// TIA Portal V18 program export: 8 tag tables, 0 data types, 0 data blocks, 7 code blocks (in call order from the OBs), 0 instance data blocks

VAR_GLOBAL   // PLC tag table "Default tag table"
   System_Byte AT %MB1 : Byte;
   FirstScan AT %M1.0 : Bool;
   DiagStatusUpdate AT %M1.1 : Bool;
   AlwaysTRUE AT %M1.2 : Bool;
   AlwaysFALSE AT %M1.3 : Bool;
   Clock_Byte AT %MB0 : Byte;
   Clock_10Hz AT %M0.0 : Bool;
   Clock_5Hz AT %M0.1 : Bool;
   "Clock_2.5Hz" AT %M0.2 : Bool;
   Clock_2Hz AT %M0.3 : Bool;
   "Clock_1.25Hz" AT %M0.4 : Bool;
   Clock_1Hz AT %M0.5 : Bool;
   "Clock_0.625Hz" AT %M0.6 : Bool;
   "Clock_0.5Hz" AT %M0.7 : Bool;
   PTRIG AT %M2.0 : Bool;
   PTRIG2 AT %M2.1 : Bool;
END_VAR

VAR_GLOBAL   // PLC tag table "INPUT"
   I_Mode AT %I0.0 : Bool;   // Switch chế độ 1 auto, 0 manu
   I_CB_Cao AT %I0.1 : Bool;   // Cảm biến sản phẩm cao
   I_CB_Trung_Binh AT %I0.2 : Bool;   // Cảm biến sản phẩm trung bình
   I_CB_Thap AT %I0.3 : Bool;   // Cảm biến sản phẩm thấp
   I_BT AT %I0.4 : Bool;   // Chạy/Dừng động cơ băng tải
   I_Xylanh_Cao AT %I0.5 : Bool;   // Đóng/mở xi lanh sản phẩm cao
   I_Xylanh_TB AT %I0.6 : Bool;   // Đóng/mở xi lanh sản phẩm trung bình
END_VAR

VAR_GLOBAL   // PLC tag table "INPUT_M"
   M_Mode AT %M10.0 : Bool;   // Switch chế độ 1 auto, 0 manu
   M_CB_Cao AT %M10.1 : Bool;   // Cảm biến sản phẩm cao
   M_CB_Trung_Binh AT %M10.2 : Bool;   // Cảm biến sản phẩm trung bình
   M_CB_Thap AT %M10.3 : Bool;   // Cảm biến sản phẩm thấp
   M_BT AT %M10.4 : Bool;   // Chạy/Dừng động cơ băng tải
   M_Xylanh_Cao AT %M10.5 : Bool;   // Đóng/mở xi lanh sản phẩm cao
   M_Xylanh_TB AT %M10.6 : Bool;   // Đóng/mở xi lanh sản phẩm trung bình
END_VAR

VAR_GLOBAL   // PLC tag table "OUTPUT"
   Q_lamp_Auto AT %Q0.0 : Bool;   // Đèn chế độ auto
   Q_lamp_Manu AT %Q0.1 : Bool;   // Đèn chế độ manu
   Q_BT AT %Q0.2 : Bool;   // Băng tải phân loại
   Q_Xylanh_Cao AT %Q0.3 : Bool;   // Xi lanh đẩy sản phẩm cao
   Q_Xylanh_TB AT %Q0.4 : Bool;   // Xi lanh đẩy sản phẩm trung bình
END_VAR

VAR_GLOBAL   // PLC tag table "PTRIG"
   P1 AT %M330.0 : Bool;
   P2 AT %M330.1 : Bool;
   P3 AT %M330.2 : Bool;
   P4 AT %M330.3 : Bool;
   P5 AT %M330.4 : Bool;
   P6 AT %M330.5 : Bool;
   P7 AT %M330.6 : Bool;
   P8 AT %M330.7 : Bool;
   P9 AT %M331.0 : Bool;
   P10 AT %M331.1 : Bool;
   P11 AT %M331.2 : Bool;
END_VAR

VAR_GLOBAL   // PLC tag table "SO_NGUYEN"
   Act_Count_Cao AT %MW200 : Int;   // Bộ đếm số sản phẩm trọng lượng nhẹ
   Act_Count_TB AT %MW202 : Int;   // Bộ đếm số sản phẩm trọng lượng trung bình
   Act_Count_Thap AT %MW204 : Int;   // Bộ đếm số sản phẩm trọng lượng nặng
   Simu_VT_SP AT %MW206 : Int;   // Mô phỏng vị trí sản phẩm
   Simu_Type_SP AT %MW208 : Int;   // Mô phỏng loại sản phẩm
END_VAR

VAR_GLOBAL   // PLC tag table "TAG"
   Start AT %I0.0 : Bool;   // Nút nhấn Start
   Stop AT %I0.1 : Bool;   // Nút nhấn Stop
   Lamp AT %Q0.0 : Bool;   // Đèn hệ thống làm việc
   Sensor_Temperature AT %IW64 : Int;   // Cảm biến nhiệt độ
   QW_SSR AT %QW64 : Int;   // Đầu ra analog điều khiển SSR
   HMI_Start AT %M10.0 : Bool;   // Nút nhấn start trên Scada
   HMI_Stop AT %M10.1 : Bool;   // Nút nhấn Stop trên Scada
   HMI_Simulation AT %M10.2 : Bool;   // Nút mô phỏng tín hiệu nhiệt độ trên Scada
   HMI_Simu_Temperature AT %MW100 : Int;   // Mô phỏng nhiệt độ trên HMI
   HMI_Setting_Temperature AT %MD200 : Real;   // Cài đặt nhiệt độ cho máy sấy
   HMI_TT_Temperature AT %MD204 : Real;   // Nhiệt độ thực tế máy sấy
END_VAR

VAR_GLOBAL   // PLC tag table "TRUNGGIAN"
   Q_Auto_BT AT %M20.0 : Bool;   // Băng tải phân loại
   Q_Auto_Xylanh_Cao AT %M20.1 : Bool;   // Xi lanh đẩy sản phẩm cao
   Q_Auto_Xylanh_TB AT %M20.2 : Bool;   // Xi lanh đẩy sản phẩm trung bình
   Q_Manu_BT AT %M30.0 : Bool;   // Băng tải phân loại
   Q_Manu_Xylanh_Cao AT %M30.1 : Bool;   // Xi lanh đẩy sản phẩm cao
   Q_Manu_Xylanh_TB AT %M30.2 : Bool;   // Xi lanh đẩy sản phẩm trung bình
   M_Simulation AT %M5.0 : Bool;   // Nút mô phỏng trên scada
   M_Reset AT %M5.1 : Bool;   // Nút reset
   SIMU_CB_CAO AT %M5.2 : Bool;   // Mô phỏng cảm biến cao
   SIMU_CB_TB AT %M5.3 : Bool;   // Mô phỏng cảm biến trung bình
   SIMU_CB_THAP AT %M5.4 : Bool;   // Mô phỏng cảm biến thấp
END_VAR

ORGANIZATION_BLOCK "Main"   // OB1, LAD, ProgramCycle
TITLE = "Main Program Sweep (Cycle)"
{ S7_Optimized_Access := 'TRUE' }
VERSION : 0.1
// stored: AutoNumber true, IsIECCheckEnabled false, SetENOAutomatically false
   VAR_INPUT
      Initial_Call : Bool;   // Initial call of this OB
      Remanence : Bool;   // =True, if remanent data are available
   END_VAR
   VAR_TEMP
      TG_ND : Int;
      TG_ND1 : Real;
   END_VAR
BEGIN

REGION Network 1: Điều khiển đèn làm việc
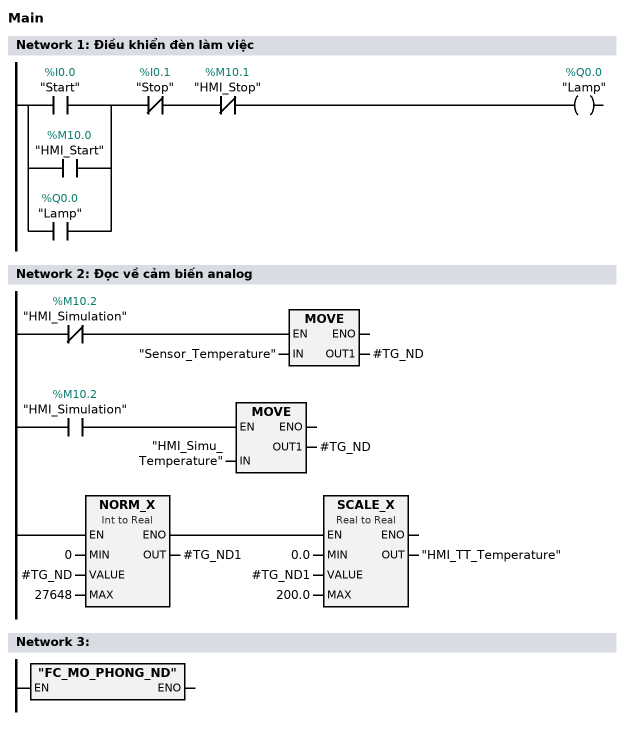
   RUNG wire#powerrail
      Contact( "Start" )
      wire#w1
      I_Contact( "Stop" )
      I_Contact( "HMI_Stop" )
      Coil( "Lamp" )
   END_RUNG
   RUNG wire#powerrail
      Contact( "HMI_Start" )
   END_RUNG wire#w1
   RUNG wire#powerrail
      Contact( "Lamp" )
   END_RUNG wire#w1
   // the same network as SCL:
   "Lamp" := ("Start" OR "HMI_Start" OR "Lamp") AND NOT "Stop" AND NOT "HMI_Stop";
END_REGION

REGION Network 2: Đọc về cảm biến analog
   RUNG wire#powerrail
      I_Contact( "HMI_Simulation" )
      Move(in := "Sensor_Temperature", out1 => #TG_ND)
   END_RUNG
   RUNG wire#powerrail
      Contact( "HMI_Simulation" )
      Move(in := "HMI_Simu_Temperature", out1 => #TG_ND)
   END_RUNG
   RUNG wire#powerrail
      { S7_Templates := "[SrcType := Int, DestType := Real]" } Normalize(min := 0, value := #TG_ND, max := 27648, out => #TG_ND1)
      { S7_Templates := "[SrcType := Real, DestType := Real]" } Scale(min := 0.0, value := #TG_ND1, max := 200.0, out => "HMI_TT_Temperature")
   END_RUNG
   // the same network as SCL:
   IF NOT "HMI_Simulation" THEN #TG_ND := "Sensor_Temperature"; END_IF;
   IF "HMI_Simulation" THEN #TG_ND := "HMI_Simu_Temperature"; END_IF;
   #TG_ND1 := NORM_X(MIN := 0, VALUE := #TG_ND, MAX := 27648);
   "HMI_TT_Temperature" := SCALE_X(MIN := 0.0, VALUE := #TG_ND1, MAX := 200.0);
END_REGION

REGION Network 3
   RUNG wire#powerrail
      "FC_MO_PHONG_ND"()
   END_RUNG
   // the same network as SCL:
   "FC_MO_PHONG_ND"();
END_REGION
END_ORGANIZATION_BLOCK

FUNCTION "FC_MO_PHONG_ND" : Void   // FC1, LAD
{ S7_Optimized_Access := 'TRUE' }
VERSION : 0.1
// stored: AutoNumber true, IsIECCheckEnabled false, SetENOAutomatically false, UDAEnableTagReadback false
   VAR_TEMP   // added for the SCL form of the ladder/FBD networks
      _w1 : Bool;
      _w2 : Bool;
      _w3 : Bool;
      _w4 : Bool;
   END_VAR
BEGIN

REGION Network 1
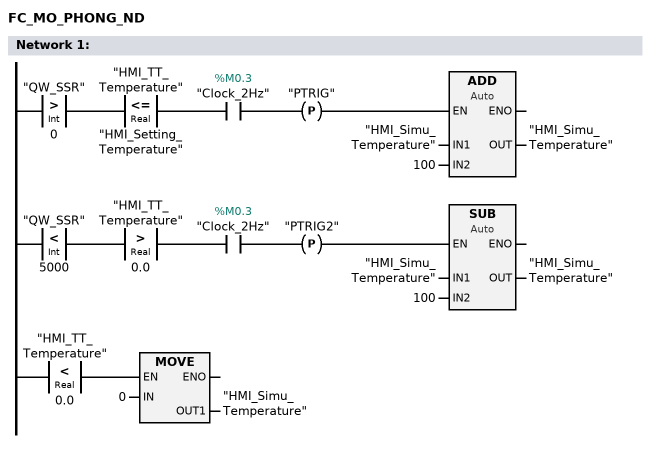
   RUNG wire#powerrail
      { S7_Templates := "SrcType := Int" } GT_Contact(in1 := "QW_SSR", in2 := 0)
      { S7_Templates := "SrcType := Real" } LE_Contact(in1 := "HMI_TT_Temperature", in2 := "HMI_Setting_Temperature")
      Contact( "Clock_2Hz" )
      P_Trig( "PTRIG" )
      Add(in1 := "HMI_Simu_Temperature", in2 := 100, out => "HMI_Simu_Temperature")
   END_RUNG
   RUNG wire#powerrail
      { S7_Templates := "SrcType := Int" } LT_Contact(in1 := "QW_SSR", in2 := 5000)
      { S7_Templates := "SrcType := Real" } GT_Contact(in1 := "HMI_TT_Temperature", in2 := 0.0)
      Contact( "Clock_2Hz" )
      P_Trig( "PTRIG2" )
      Sub(in1 := "HMI_Simu_Temperature", in2 := 100, out => "HMI_Simu_Temperature")
   END_RUNG
   RUNG wire#powerrail
      { S7_Templates := "SrcType := Real" } LT_Contact(in1 := "HMI_TT_Temperature", in2 := 0.0)
      Move(in := 0, out1 => "HMI_Simu_Temperature")
   END_RUNG
   // the same network as SCL:
   #_w1 := ("QW_SSR" > 0) AND ("HMI_TT_Temperature" <= "HMI_Setting_Temperature") AND "Clock_2Hz";
   #_w2 := #_w1 AND NOT "PTRIG";   // rising edge
   "PTRIG" := #_w1;
   IF #_w2 THEN "HMI_Simu_Temperature" := "HMI_Simu_Temperature" + 100; END_IF;
   #_w3 := ("QW_SSR" < 5000) AND ("HMI_TT_Temperature" > 0.0) AND "Clock_2Hz";
   #_w4 := #_w3 AND NOT "PTRIG2";   // rising edge
   "PTRIG2" := #_w3;
   IF #_w4 THEN "HMI_Simu_Temperature" := "HMI_Simu_Temperature" - 100; END_IF;
   IF "HMI_TT_Temperature" < 0.0 THEN "HMI_Simu_Temperature" := 0; END_IF;
END_REGION
END_FUNCTION

ORGANIZATION_BLOCK "Cyclic interrupt"   // OB30, LAD, CyclicInterrupt
{ S7_Optimized_Access := 'TRUE' }
VERSION : 0.1
// stored: AutoNumber true, IsIECCheckEnabled false, SetENOAutomatically false
   VAR_INPUT
      Initial_Call : Bool;   // Initial call of this OB
      Event_Count : Int;   // Events discarded
   END_VAR
BEGIN

REGION Network 1
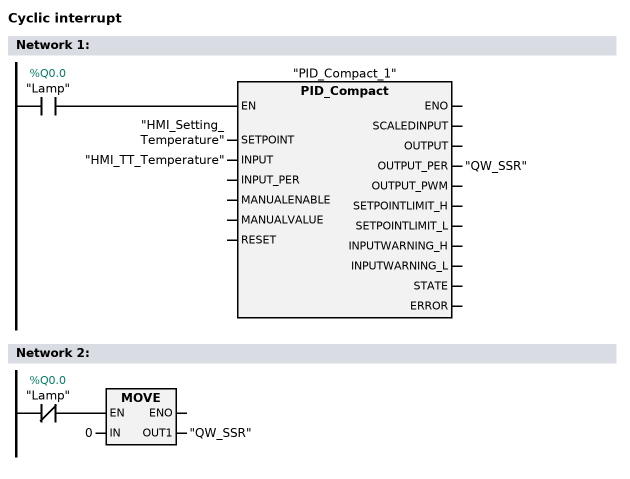
   RUNG wire#powerrail
      Contact( "Lamp" )
      "PID_Compact_1".PID_Compact(Setpoint := "HMI_Setting_Temperature", Input := "HMI_TT_Temperature", Input_PER :=, ManualEnable :=, ManualValue :=, Reset :=, ScaledInput =>, Output =>, Output_PER => "QW_SSR", Output_PWM =>, SetpointLimit_H =>, SetpointLimit_L =>, InputWarning_H =>, InputWarning_L =>, State =>, Error =>)
   END_RUNG
   // the same network as SCL:
   IF "Lamp" THEN
       "PID_Compact_1"(Setpoint := "HMI_Setting_Temperature", Input := "HMI_TT_Temperature", Output_PER => "QW_SSR");   // PID_Compact
   END_IF;
END_REGION

REGION Network 2
   RUNG wire#powerrail
      I_Contact( "Lamp" )
      Move(in := 0, out1 => "QW_SSR")
   END_RUNG
   // the same network as SCL:
   IF NOT "Lamp" THEN "QW_SSR" := 0; END_IF;
END_REGION
END_ORGANIZATION_BLOCK

FUNCTION "FC_AUTO_MODE" : Void   // FC2, LAD
{ S7_Optimized_Access := 'TRUE' }
VERSION : 0.1
// stored: AutoNumber true, IsIECCheckEnabled false, SetENOAutomatically false, UDAEnableTagReadback false
   VAR_TEMP   // added for the SCL form of the ladder/FBD networks
      _w1 : Bool;
      _w2 : Bool;
      _w3 : Bool;
      _w4 : Bool;
      _w5 : Bool;
      _w6 : Bool;
   END_VAR
BEGIN

REGION Network 1: RESET CÁC BỘ ĐẾM VỀ 0
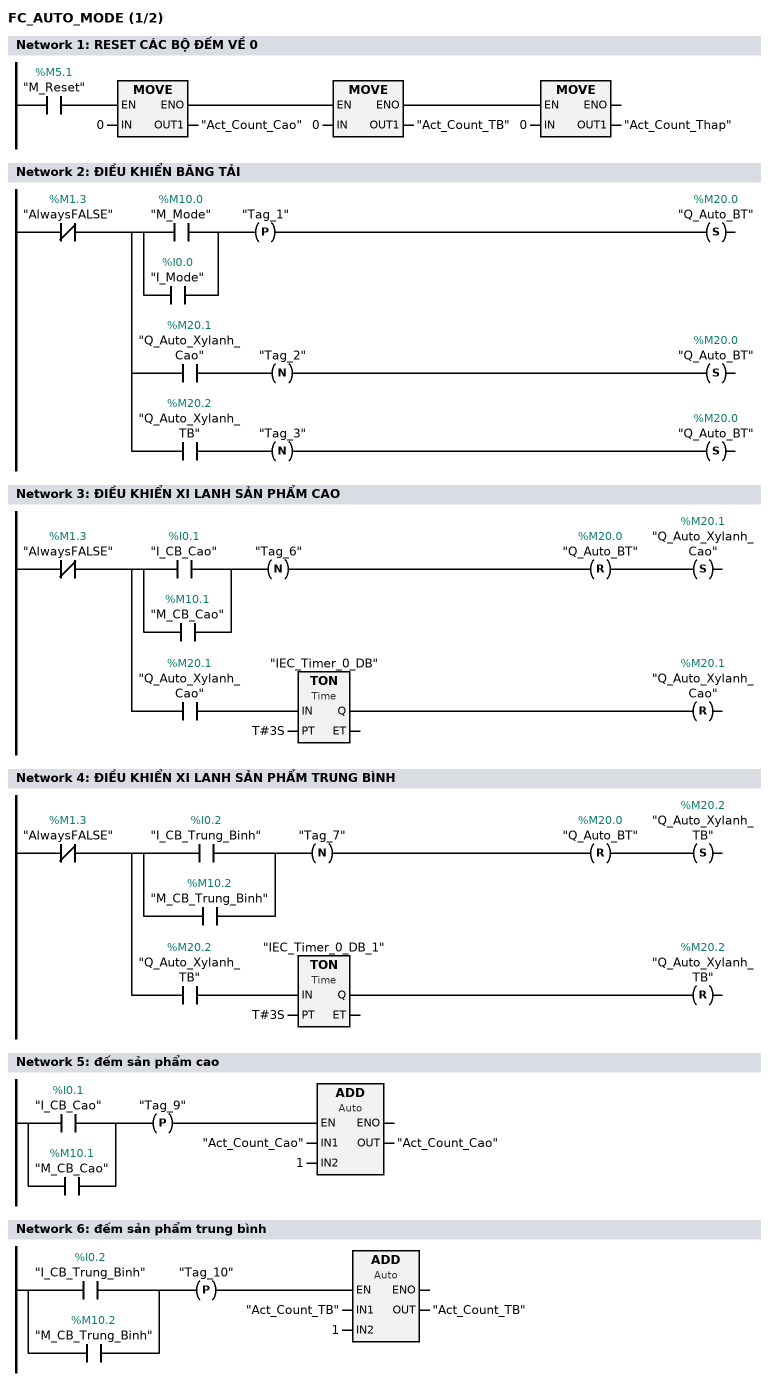
   RUNG wire#powerrail
      Contact( "M_Reset" )
      Move(in := 0, out1 => "Act_Count_Cao")
      Move(in := 0, out1 => "Act_Count_TB")
      Move(in := 0, out1 => "Act_Count_Thap")
   END_RUNG
   // the same network as SCL:
   IF "M_Reset" THEN
       "Act_Count_Cao" := 0;
       "Act_Count_TB" := 0;
       "Act_Count_Thap" := 0;
   END_IF;
END_REGION

REGION Network 2: ĐIỀU KHIỂN BĂNG TẢI
   RUNG wire#powerrail
      I_Contact( "AlwaysFALSE" )
      wire#w1
      Contact( "M_Mode" )
      wire#w2
      P_Trig( "Tag_1" )
      S_Coil( "Q_Auto_BT" )
   END_RUNG
   RUNG wire#w1
      Contact( "I_Mode" )
   END_RUNG wire#w2
   RUNG wire#w1
      Contact( "Q_Auto_Xylanh_Cao" )
      N_Trig( "Tag_2" )
      S_Coil( "Q_Auto_BT" )
   END_RUNG
   RUNG wire#w1
      Contact( "Q_Auto_Xylanh_TB" )
      N_Trig( "Tag_3" )
      S_Coil( "Q_Auto_BT" )
   END_RUNG
   // the same network as SCL:
   #_w1 := NOT "AlwaysFALSE" AND ("M_Mode" OR "I_Mode");
   #_w2 := #_w1 AND NOT "Tag_1";   // rising edge
   "Tag_1" := #_w1;
   IF #_w2 THEN "Q_Auto_BT" := TRUE; END_IF;
   #_w3 := NOT "AlwaysFALSE" AND "Q_Auto_Xylanh_Cao";
   #_w4 := NOT #_w3 AND "Tag_2";   // falling edge
   "Tag_2" := #_w3;
   IF #_w4 THEN "Q_Auto_BT" := TRUE; END_IF;
   #_w5 := NOT "AlwaysFALSE" AND "Q_Auto_Xylanh_TB";
   #_w6 := NOT #_w5 AND "Tag_3";   // falling edge
   "Tag_3" := #_w5;
   IF #_w6 THEN "Q_Auto_BT" := TRUE; END_IF;
END_REGION

REGION Network 3: ĐIỀU KHIỂN XI LANH SẢN PHẨM CAO
   RUNG wire#powerrail
      I_Contact( "AlwaysFALSE" )
      wire#w1
      Contact( "I_CB_Cao" )
      wire#w2
      N_Trig( "Tag_6" )
      R_Coil( "Q_Auto_BT" )
      S_Coil( "Q_Auto_Xylanh_Cao" )
   END_RUNG
   RUNG wire#w1
      Contact( "M_CB_Cao" )
   END_RUNG wire#w2
   RUNG wire#w1
      Contact( "Q_Auto_Xylanh_Cao" )
      { S7_Templates := "time_type := Time" } "IEC_Timer_0_DB".TON(pt := T#3S, et =>)
      R_Coil( "Q_Auto_Xylanh_Cao" )
   END_RUNG
   // the same network as SCL:
   #_w1 := NOT "AlwaysFALSE" AND ("I_CB_Cao" OR "M_CB_Cao");
   #_w2 := NOT #_w1 AND "Tag_6";   // falling edge
   "Tag_6" := #_w1;
   IF #_w2 THEN
       "Q_Auto_BT" := FALSE;
       "Q_Auto_Xylanh_Cao" := TRUE;
   END_IF;
   "IEC_Timer_0_DB".TON(IN := NOT "AlwaysFALSE" AND "Q_Auto_Xylanh_Cao", PT := T#3S);
   IF "IEC_Timer_0_DB".Q THEN "Q_Auto_Xylanh_Cao" := FALSE; END_IF;
END_REGION

REGION Network 4: ĐIỀU KHIỂN XI LANH SẢN PHẨM TRUNG BÌNH
   RUNG wire#powerrail
      I_Contact( "AlwaysFALSE" )
      wire#w1
      Contact( "I_CB_Trung_Binh" )
      wire#w2
      N_Trig( "Tag_7" )
      R_Coil( "Q_Auto_BT" )
      S_Coil( "Q_Auto_Xylanh_TB" )
   END_RUNG
   RUNG wire#w1
      Contact( "M_CB_Trung_Binh" )
   END_RUNG wire#w2
   RUNG wire#w1
      Contact( "Q_Auto_Xylanh_TB" )
      { S7_Templates := "time_type := Time" } "IEC_Timer_0_DB_1".TON(pt := T#3S, et =>)
      R_Coil( "Q_Auto_Xylanh_TB" )
   END_RUNG
   // the same network as SCL:
   #_w1 := NOT "AlwaysFALSE" AND ("I_CB_Trung_Binh" OR "M_CB_Trung_Binh");
   #_w2 := NOT #_w1 AND "Tag_7";   // falling edge
   "Tag_7" := #_w1;
   IF #_w2 THEN
       "Q_Auto_BT" := FALSE;
       "Q_Auto_Xylanh_TB" := TRUE;
   END_IF;
   "IEC_Timer_0_DB_1".TON(IN := NOT "AlwaysFALSE" AND "Q_Auto_Xylanh_TB", PT := T#3S);
   IF "IEC_Timer_0_DB_1".Q THEN "Q_Auto_Xylanh_TB" := FALSE; END_IF;
END_REGION

REGION Network 5: đếm sản phẩm cao
   RUNG wire#powerrail
      Contact( "I_CB_Cao" )
      wire#w1
      P_Trig( "Tag_9" )
      Add(in1 := "Act_Count_Cao", in2 := 1, out => "Act_Count_Cao")
   END_RUNG
   RUNG wire#powerrail
      Contact( "M_CB_Cao" )
   END_RUNG wire#w1
   // the same network as SCL:
   #_w1 := "I_CB_Cao" OR "M_CB_Cao";
   #_w2 := #_w1 AND NOT "Tag_9";   // rising edge
   "Tag_9" := #_w1;
   IF #_w2 THEN "Act_Count_Cao" := "Act_Count_Cao" + 1; END_IF;
END_REGION

REGION Network 6: đếm sản phẩm trung bình
   RUNG wire#powerrail
      Contact( "I_CB_Trung_Binh" )
      wire#w1
      P_Trig( "Tag_10" )
      Add(in1 := "Act_Count_TB", in2 := 1, out => "Act_Count_TB")
   END_RUNG
   RUNG wire#powerrail
      Contact( "M_CB_Trung_Binh" )
   END_RUNG wire#w1
   // the same network as SCL:
   #_w1 := "I_CB_Trung_Binh" OR "M_CB_Trung_Binh";
   #_w2 := #_w1 AND NOT "Tag_10";   // rising edge
   "Tag_10" := #_w1;
   IF #_w2 THEN "Act_Count_TB" := "Act_Count_TB" + 1; END_IF;
END_REGION

REGION Network 7: đếm sản phẩm thấp
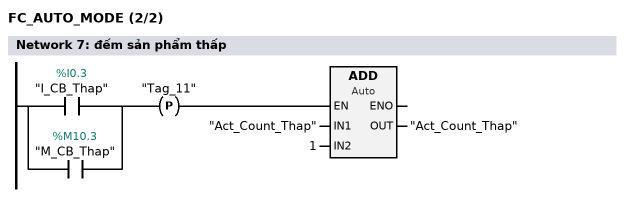
   RUNG wire#powerrail
      Contact( "I_CB_Thap" )
      wire#w1
      P_Trig( "Tag_11" )
      Add(in1 := "Act_Count_Thap", in2 := 1, out => "Act_Count_Thap")
   END_RUNG
   RUNG wire#powerrail
      Contact( "M_CB_Thap" )
   END_RUNG wire#w1
   // the same network as SCL:
   #_w1 := "I_CB_Thap" OR "M_CB_Thap";
   #_w2 := #_w1 AND NOT "Tag_11";   // rising edge
   "Tag_11" := #_w1;
   IF #_w2 THEN "Act_Count_Thap" := "Act_Count_Thap" + 1; END_IF;
END_REGION
END_FUNCTION

FUNCTION "FC_MANUAL_MODE" : Void   // FC1, LAD
{ S7_Optimized_Access := 'TRUE' }
VERSION : 0.1
// stored: AutoNumber true, IsIECCheckEnabled false, SetENOAutomatically false, UDAEnableTagReadback false
BEGIN

REGION Network 1: BĂNG TẢI
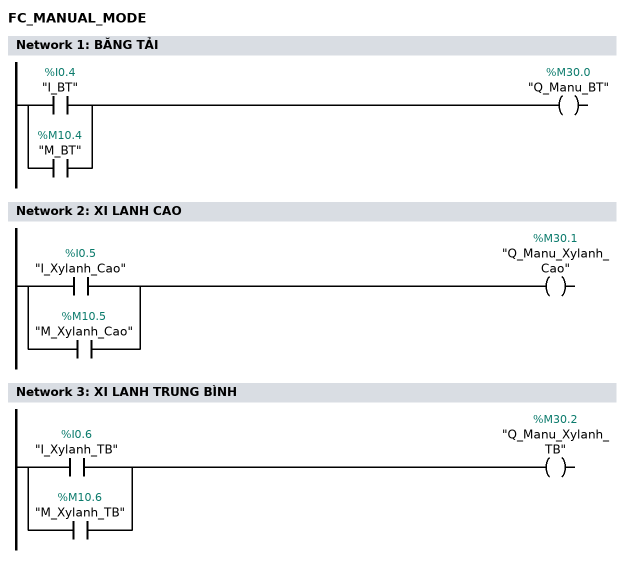
   RUNG wire#powerrail
      Contact( "I_BT" )
      wire#w1
      Coil( "Q_Manu_BT" )
   END_RUNG
   RUNG wire#powerrail
      Contact( "M_BT" )
   END_RUNG wire#w1
   // the same network as SCL:
   "Q_Manu_BT" := "I_BT" OR "M_BT";
END_REGION

REGION Network 2: XI LANH CAO
   RUNG wire#powerrail
      Contact( "I_Xylanh_Cao" )
      wire#w1
      Coil( "Q_Manu_Xylanh_Cao" )
   END_RUNG
   RUNG wire#powerrail
      Contact( "M_Xylanh_Cao" )
   END_RUNG wire#w1
   // the same network as SCL:
   "Q_Manu_Xylanh_Cao" := "I_Xylanh_Cao" OR "M_Xylanh_Cao";
END_REGION

REGION Network 3: XI LANH TRUNG BÌNH
   RUNG wire#powerrail
      Contact( "I_Xylanh_TB" )
      wire#w1
      Coil( "Q_Manu_Xylanh_TB" )
   END_RUNG
   RUNG wire#powerrail
      Contact( "M_Xylanh_TB" )
   END_RUNG wire#w1
   // the same network as SCL:
   "Q_Manu_Xylanh_TB" := "I_Xylanh_TB" OR "M_Xylanh_TB";
END_REGION
END_FUNCTION

FUNCTION "FC_OUTPUT" : Void   // FC3, LAD
{ S7_Optimized_Access := 'TRUE' }
VERSION : 0.1
// stored: AutoNumber true, IsIECCheckEnabled false, SetENOAutomatically false, UDAEnableTagReadback false
BEGIN

REGION Network 1: BĂNG TẢI
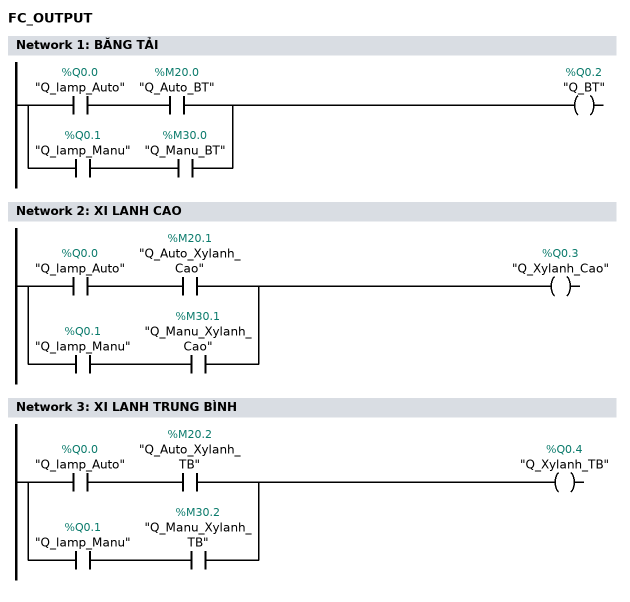
   RUNG wire#powerrail
      Contact( "Q_lamp_Auto" )
      Contact( "Q_Auto_BT" )
      wire#w1
      Coil( "Q_BT" )
   END_RUNG
   RUNG wire#powerrail
      Contact( "Q_lamp_Manu" )
      Contact( "Q_Manu_BT" )
   END_RUNG wire#w1
   // the same network as SCL:
   "Q_BT" := ("Q_lamp_Auto" AND "Q_Auto_BT") OR ("Q_lamp_Manu" AND "Q_Manu_BT");
END_REGION

REGION Network 2: XI LANH CAO
   RUNG wire#powerrail
      Contact( "Q_lamp_Auto" )
      Contact( "Q_Auto_Xylanh_Cao" )
      wire#w1
      Coil( "Q_Xylanh_Cao" )
   END_RUNG
   RUNG wire#powerrail
      Contact( "Q_lamp_Manu" )
      Contact( "Q_Manu_Xylanh_Cao" )
   END_RUNG wire#w1
   // the same network as SCL:
   "Q_Xylanh_Cao" := ("Q_lamp_Auto" AND "Q_Auto_Xylanh_Cao") OR ("Q_lamp_Manu" AND "Q_Manu_Xylanh_Cao");
END_REGION

REGION Network 3: XI LANH TRUNG BÌNH
   RUNG wire#powerrail
      Contact( "Q_lamp_Auto" )
      Contact( "Q_Auto_Xylanh_TB" )
      wire#w1
      Coil( "Q_Xylanh_TB" )
   END_RUNG
   RUNG wire#powerrail
      Contact( "Q_lamp_Manu" )
      Contact( "Q_Manu_Xylanh_TB" )
   END_RUNG wire#w1
   // the same network as SCL:
   "Q_Xylanh_TB" := ("Q_lamp_Auto" AND "Q_Auto_Xylanh_TB") OR ("Q_lamp_Manu" AND "Q_Manu_Xylanh_TB");
END_REGION
END_FUNCTION

FUNCTION "FC_SIMULATION" : Void   // FC4, LAD
{ S7_Optimized_Access := 'TRUE' }
VERSION : 0.1
// stored: AutoNumber true, IsIECCheckEnabled false, SetENOAutomatically false, UDAEnableTagReadback false
   VAR_TEMP   // added for the SCL form of the ladder/FBD networks
      _w1 : Bool;
      _w2 : Bool;
      _w3 : Bool;
      _w4 : Bool;
      _w5 : Bool;
      _w6 : Bool;
   END_VAR
BEGIN

REGION Network 1: KHỞI ĐỘNG LÀ CHẠY SIMU CẢM BIẾN Cao LUÔN
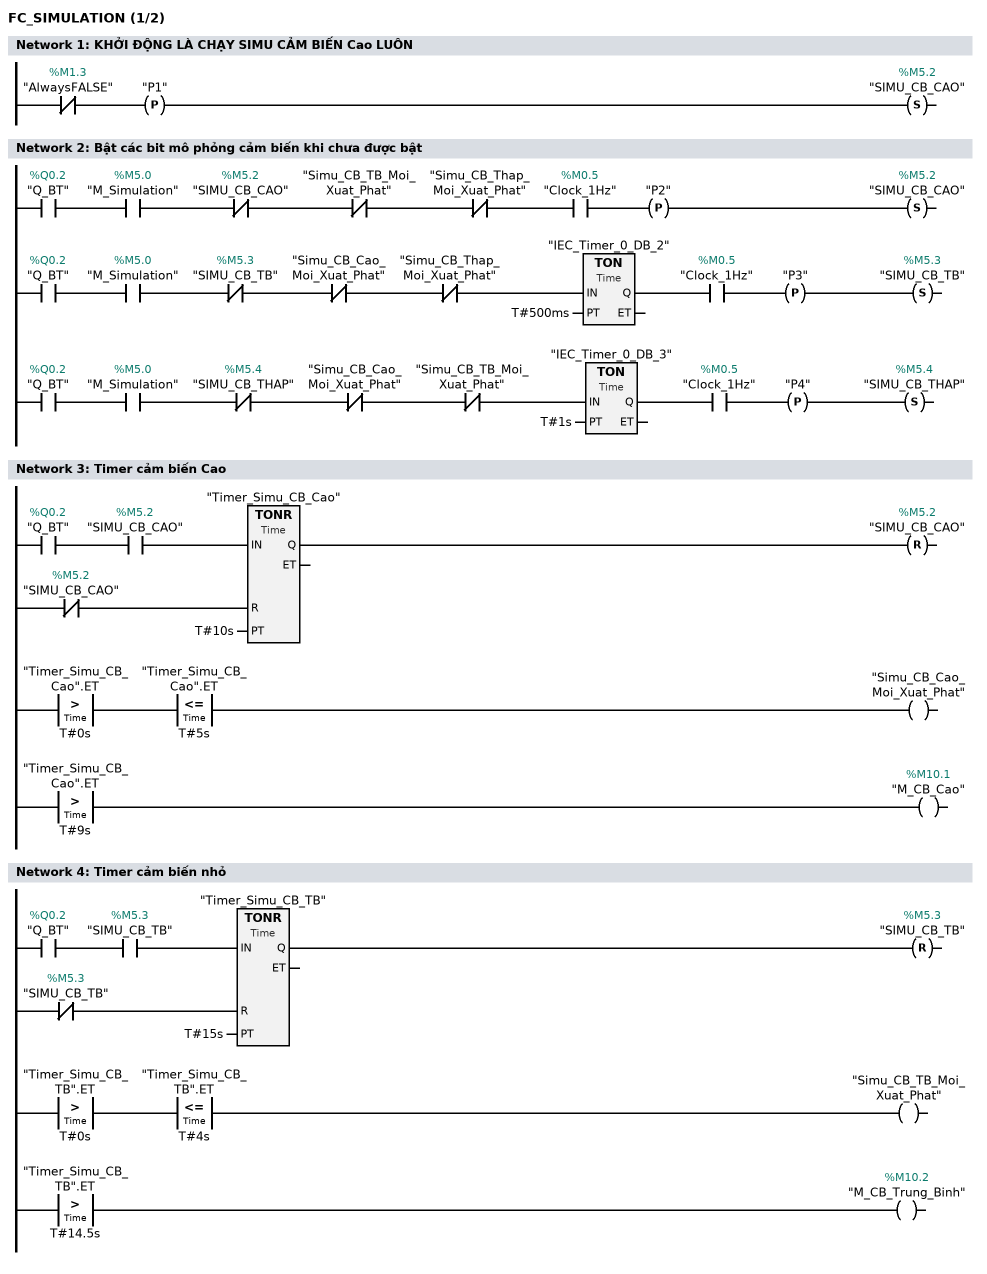
   RUNG wire#powerrail
      I_Contact( "AlwaysFALSE" )
      P_Trig( "P1" )
      S_Coil( "SIMU_CB_CAO" )
   END_RUNG
   // the same network as SCL:
   #_w1 := NOT "AlwaysFALSE" AND NOT "P1";   // rising edge
   "P1" := NOT "AlwaysFALSE";
   IF #_w1 THEN "SIMU_CB_CAO" := TRUE; END_IF;
END_REGION

REGION Network 2: Bật các bit mô phỏng cảm biến khi chưa được bật
   RUNG wire#powerrail
      Contact( "Q_BT" )
      Contact( "M_Simulation" )
      I_Contact( "SIMU_CB_CAO" )
      I_Contact( "Simu_CB_TB_Moi_Xuat_Phat" )
      I_Contact( "Simu_CB_Thap_Moi_Xuat_Phat" )
      Contact( "Clock_1Hz" )
      P_Trig( "P2" )
      S_Coil( "SIMU_CB_CAO" )
   END_RUNG
   RUNG wire#powerrail
      Contact( "Q_BT" )
      Contact( "M_Simulation" )
      I_Contact( "SIMU_CB_TB" )
      I_Contact( "Simu_CB_Cao_Moi_Xuat_Phat" )
      I_Contact( "Simu_CB_Thap_Moi_Xuat_Phat" )
      { S7_Templates := "time_type := Time" } "IEC_Timer_0_DB_2".TON(pt := T#500ms, et =>)
      Contact( "Clock_1Hz" )
      P_Trig( "P3" )
      S_Coil( "SIMU_CB_TB" )
   END_RUNG
   RUNG wire#powerrail
      Contact( "Q_BT" )
      Contact( "M_Simulation" )
      I_Contact( "SIMU_CB_THAP" )
      I_Contact( "Simu_CB_Cao_Moi_Xuat_Phat" )
      I_Contact( "Simu_CB_TB_Moi_Xuat_Phat" )
      { S7_Templates := "time_type := Time" } "IEC_Timer_0_DB_3".TON(pt := T#1s, et =>)
      Contact( "Clock_1Hz" )
      P_Trig( "P4" )
      S_Coil( "SIMU_CB_THAP" )
   END_RUNG
   // the same network as SCL:
   #_w1 := "Q_BT" AND "M_Simulation" AND NOT "SIMU_CB_CAO" AND NOT "Simu_CB_TB_Moi_Xuat_Phat" AND NOT "Simu_CB_Thap_Moi_Xuat_Phat" AND "Clock_1Hz";
   #_w2 := #_w1 AND NOT "P2";   // rising edge
   "P2" := #_w1;
   IF #_w2 THEN "SIMU_CB_CAO" := TRUE; END_IF;
   "IEC_Timer_0_DB_2".TON(IN := "Q_BT" AND "M_Simulation" AND NOT "SIMU_CB_TB" AND NOT "Simu_CB_Cao_Moi_Xuat_Phat" AND NOT "Simu_CB_Thap_Moi_Xuat_Phat",
                          PT := T#500ms);
   #_w3 := "IEC_Timer_0_DB_2".Q AND "Clock_1Hz";
   #_w4 := #_w3 AND NOT "P3";   // rising edge
   "P3" := #_w3;
   IF #_w4 THEN "SIMU_CB_TB" := TRUE; END_IF;
   "IEC_Timer_0_DB_3".TON(IN := "Q_BT" AND "M_Simulation" AND NOT "SIMU_CB_THAP" AND NOT "Simu_CB_Cao_Moi_Xuat_Phat" AND NOT "Simu_CB_TB_Moi_Xuat_Phat",
                          PT := T#1s);
   #_w5 := "IEC_Timer_0_DB_3".Q AND "Clock_1Hz";
   #_w6 := #_w5 AND NOT "P4";   // rising edge
   "P4" := #_w5;
   IF #_w6 THEN "SIMU_CB_THAP" := TRUE; END_IF;
END_REGION

REGION Network 3: Timer cảm biến Cao
   RUNG wire#powerrail
      Contact( "Q_BT" )
      Contact( "SIMU_CB_CAO" )
      { S7_Templates := "time_type := Time" } "Timer_Simu_CB_Cao".TONR(r := wire#w1, pt := T#10s, et =>)
      R_Coil( "SIMU_CB_CAO" )
   END_RUNG
   RUNG wire#powerrail
      I_Contact( "SIMU_CB_CAO" )
   END_RUNG wire#w1
   RUNG wire#powerrail
      { S7_Templates := "SrcType := Time" } GT_Contact(in1 := "Timer_Simu_CB_Cao".ET, in2 := T#0s)
      { S7_Templates := "SrcType := Time" } LE_Contact(in1 := "Timer_Simu_CB_Cao".ET, in2 := T#5s)
      Coil( "Simu_CB_Cao_Moi_Xuat_Phat" )
   END_RUNG
   RUNG wire#powerrail
      { S7_Templates := "SrcType := Time" } GT_Contact(in1 := "Timer_Simu_CB_Cao".ET, in2 := T#9s)
      Coil( "M_CB_Cao" )
   END_RUNG
   // the same network as SCL:
   "Timer_Simu_CB_Cao".TONR(IN := "Q_BT" AND "SIMU_CB_CAO", R := NOT "SIMU_CB_CAO", PT := T#10s);
   IF "Timer_Simu_CB_Cao".Q THEN "SIMU_CB_CAO" := FALSE; END_IF;
   "Simu_CB_Cao_Moi_Xuat_Phat" := ("Timer_Simu_CB_Cao".ET > T#0s) AND ("Timer_Simu_CB_Cao".ET <= T#5s);
   "M_CB_Cao" := "Timer_Simu_CB_Cao".ET > T#9s;
END_REGION

REGION Network 4: Timer cảm biến nhỏ
   RUNG wire#powerrail
      Contact( "Q_BT" )
      Contact( "SIMU_CB_TB" )
      { S7_Templates := "time_type := Time" } "Timer_Simu_CB_TB".TONR(r := wire#w1, pt := T#15s, et =>)
      R_Coil( "SIMU_CB_TB" )
   END_RUNG
   RUNG wire#powerrail
      I_Contact( "SIMU_CB_TB" )
   END_RUNG wire#w1
   RUNG wire#powerrail
      { S7_Templates := "SrcType := Time" } GT_Contact(in1 := "Timer_Simu_CB_TB".ET, in2 := T#0s)
      { S7_Templates := "SrcType := Time" } LE_Contact(in1 := "Timer_Simu_CB_TB".ET, in2 := T#4s)
      Coil( "Simu_CB_TB_Moi_Xuat_Phat" )
   END_RUNG
   RUNG wire#powerrail
      { S7_Templates := "SrcType := Time" } GT_Contact(in1 := "Timer_Simu_CB_TB".ET, in2 := T#14.5s)
      Coil( "M_CB_Trung_Binh" )
   END_RUNG
   // the same network as SCL:
   "Timer_Simu_CB_TB".TONR(IN := "Q_BT" AND "SIMU_CB_TB", R := NOT "SIMU_CB_TB", PT := T#15s);
   IF "Timer_Simu_CB_TB".Q THEN "SIMU_CB_TB" := FALSE; END_IF;
   "Simu_CB_TB_Moi_Xuat_Phat" := ("Timer_Simu_CB_TB".ET > T#0s) AND ("Timer_Simu_CB_TB".ET <= T#4s);
   "M_CB_Trung_Binh" := "Timer_Simu_CB_TB".ET > T#14.5s;
END_REGION

REGION Network 5: Mô phỏng cảm biến trung bình
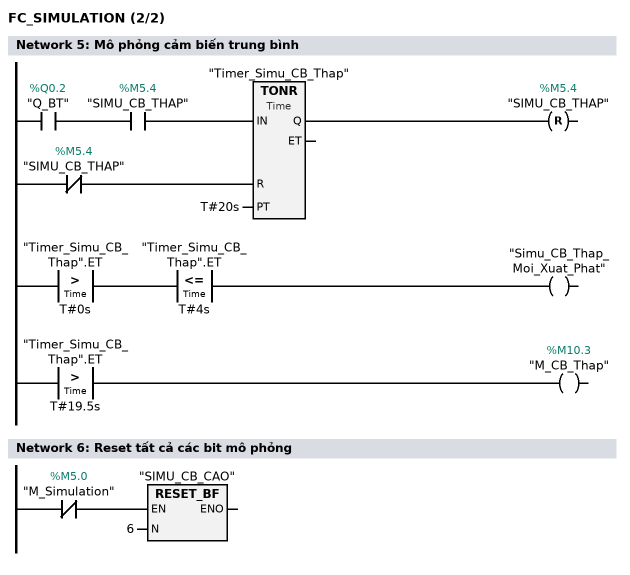
   RUNG wire#powerrail
      Contact( "Q_BT" )
      Contact( "SIMU_CB_THAP" )
      { S7_Templates := "time_type := Time" } "Timer_Simu_CB_Thap".TONR(r := wire#w1, pt := T#20s, et =>)
      R_Coil( "SIMU_CB_THAP" )
   END_RUNG
   RUNG wire#powerrail
      I_Contact( "SIMU_CB_THAP" )
   END_RUNG wire#w1
   RUNG wire#powerrail
      { S7_Templates := "SrcType := Time" } GT_Contact(in1 := "Timer_Simu_CB_Thap".ET, in2 := T#0s)
      { S7_Templates := "SrcType := Time" } LE_Contact(in1 := "Timer_Simu_CB_Thap".ET, in2 := T#4s)
      Coil( "Simu_CB_Thap_Moi_Xuat_Phat" )
   END_RUNG
   RUNG wire#powerrail
      { S7_Templates := "SrcType := Time" } GT_Contact(in1 := "Timer_Simu_CB_Thap".ET, in2 := T#19.5s)
      Coil( "M_CB_Thap" )
   END_RUNG
   // the same network as SCL:
   "Timer_Simu_CB_Thap".TONR(IN := "Q_BT" AND "SIMU_CB_THAP", R := NOT "SIMU_CB_THAP", PT := T#20s);
   IF "Timer_Simu_CB_Thap".Q THEN "SIMU_CB_THAP" := FALSE; END_IF;
   "Simu_CB_Thap_Moi_Xuat_Phat" := ("Timer_Simu_CB_Thap".ET > T#0s) AND ("Timer_Simu_CB_Thap".ET <= T#4s);
   "M_CB_Thap" := "Timer_Simu_CB_Thap".ET > T#19.5s;
END_REGION

REGION Network 6: Reset tất cả các bit mô phỏng
   // no SCL statement known for RBitfield: written as a call
   IF NOT "M_Simulation" THEN RESET_BF(operand := "SIMU_CB_CAO", n := 6); END_IF;
END_REGION
END_FUNCTION
